Universal Robots URScript: step3_0e_min_speedl_1ms_v2.script

# Step3-0E v2: minimal speedl(t=0.001) isolation with heartbeat-start gate.
# VERSION: 2026-06-08T1155HKT_STEP3_0E_MIN_SPEEDL_1MS_V2
# GENERATED_AT_LOCAL: 2026-06-08T11:55:00+0800
# BEHAVIOR: wait until the RTDE input heartbeat actually changes, then run the
# same minimal speedl(t=0.001) test. This prevents the program from consuming
# its short motion window during the benchmark's Kunwei-only baseline period.
# MOTION: stage 52 commands +X at 2 mm/s for 0.5 s, stage 53 commands -X at
# 2 mm/s for 0.5 s, so the planned round trip is about 1 mm out and 1 mm back.
# ACCELERATION: speedl acceleration a=0.100 m/s^2 = 100 mm/s^2.
# SAFETY BOUNDARY: no contact search, no force-control law, no zero/tare/config
# writes, no movel/stopl/force mode.

def codex_wait_for_fresh_heartbeat(timeout_s):
  local wait_dt = 0.002
  local t = 0.0
  local initial_heartbeat = read_input_float_register(26)
  local current_heartbeat = initial_heartbeat
  while t < timeout_s:
    current_heartbeat = read_input_float_register(26)
    write_output_float_register(26, current_heartbeat)
    write_output_float_register(34, 50.0)
    write_output_float_register(35, t)
    if read_input_float_register(27) > 0.5 and current_heartbeat != initial_heartbeat:
      return True
    end
    sync()
    t = t + wait_dt
  end
  return False
end

def codex_step3_0e_min_speedl_1ms_v2():
  local dt = 0.001
  local runtime_s = 120.0
  local zero_hold_s = 1.0
  local move_each_way_s = 0.5
  local speed_x_m_s = 0.002
  local accel_m_s2 = 0.100
  local t = 0.0
  local loop_counter = 0.0
  local stop_reason = 0.0
  local stage = 50.0

  textmsg("codex step3-0e min speedl version 2026-06-08T1155HKT_STEP3_0E_MIN_SPEEDL_1MS_V2 start speed=2mmps accel=100mmps2 t=1ms")

  if not codex_wait_for_fresh_heartbeat(30.0):
    stop_reason = 3.0
  end

  while t < runtime_s and stop_reason == 0.0:
    local normal_force = read_input_float_register(24)
    local force_norm = read_input_float_register(25)
    local heartbeat = read_input_float_register(26)
    local sensor_ok = read_input_float_register(27)
    local stop_request = read_input_float_register(28)
    local target_force_abs = read_input_float_register(29)
    local pose_now = get_actual_tcp_pose()

    local vx = 0.0
    if t < zero_hold_s:
      stage = 51.0
      vx = 0.0
    elif t < zero_hold_s + move_each_way_s:
      stage = 52.0
      vx = speed_x_m_s
    elif t < zero_hold_s + 2.0 * move_each_way_s:
      stage = 53.0
      vx = -speed_x_m_s
    else:
      stage = 54.0
      vx = 0.0
    end

    if sensor_ok < 0.5:
      stop_reason = 3.0
    elif stop_request > 0.5:
      stop_reason = 4.0
    end

    write_output_float_register(24, normal_force)
    write_output_float_register(25, force_norm)
    write_output_float_register(26, heartbeat)
    write_output_float_register(27, sensor_ok)
    write_output_float_register(28, stop_request)
    write_output_float_register(29, target_force_abs)
    write_output_float_register(30, stop_reason)
    write_output_float_register(31, pose_now[0])
    write_output_float_register(32, pose_now[1])
    write_output_float_register(33, vx)
    write_output_float_register(34, stage)
    write_output_float_register(35, loop_counter)

    speedl([vx, 0.0, 0.0, 0.0, 0.0, 0.0], accel_m_s2, dt)
    loop_counter = loop_counter + 1.0
    t = t + dt
  end

  speedl([0.0, 0.0, 0.0, 0.0, 0.0, 0.0], accel_m_s2, 0.010)
  write_output_float_register(30, stop_reason)
  textmsg("codex step3-0e min speedl version 2026-06-08T1155HKT_STEP3_0E_MIN_SPEEDL_1MS_V2 stop reason:", stop_reason)
end

codex_step3_0e_min_speedl_1ms_v2()
